TYPE ST_ShortcutConfig :
STRUCT
	TestPowerMat  						: BOOL;
END_STRUCT
END_TYPE

(* stored: Version 1.1.0.1
   DUT ST_ShortcutConfig: Id {26fa2e14-a928-012c-3abf-7a0b030ea531} *)
